{attribute 'GeneratedUsingTerminal: EP8309-0022-0021'}
{attribute addProperty BoxType "EP8309-0022-0021"}
{attribute addProperty Id "Digital_Input_X4_Pin4AT %I*BOOL1Digital_Input_X4_Pin2AT %I*BOOL1Digital_Input_X5_Pin4AT %I*BOOL1Digital_Input_X5_Pin2AT %I*BOOL1Digital_Input_X6_Pin4AT %I*BOOL1Digital_Input_X6_Pin2AT %I*BOOL1Digital_Input_X7_Pin4AT %I*BOOL1Digital_Input_X7_Pin2AT %I*BOOL1"}
{attribute addProperty CRC "1230986660"}
{attribute addProperty Size "8"}
TYPE DIG_Inputs_495F5DA4 EXTENDS InputBase_8311D824 :
STRUCT
	{attribute addProperty Name "Digital_Input_X4_Pin4"}
	Digital_Input_X4_Pin4 AT %I* : BOOL;
	{attribute addProperty Name "Digital_Input_X4_Pin2"}
	Digital_Input_X4_Pin2 AT %I* : BOOL;
	{attribute addProperty Name "Digital_Input_X5_Pin4"}
	Digital_Input_X5_Pin4 AT %I* : BOOL;
	{attribute addProperty Name "Digital_Input_X5_Pin2"}
	Digital_Input_X5_Pin2 AT %I* : BOOL;
	{attribute addProperty Name "Digital_Input_X6_Pin4"}
	Digital_Input_X6_Pin4 AT %I* : BOOL;
	{attribute addProperty Name "Digital_Input_X6_Pin2"}
	Digital_Input_X6_Pin2 AT %I* : BOOL;
	{attribute addProperty Name "Digital_Input_X7_Pin4"}
	Digital_Input_X7_Pin4 AT %I* : BOOL;
	{attribute addProperty Name "Digital_Input_X7_Pin2"}
	Digital_Input_X7_Pin2 AT %I* : BOOL;
END_STRUCT
END_TYPE

(* stored: Version 1.2.0.0, ProductVersion 3.1.4024.9
   DUT DIG_Inputs_495F5DA4: Id {d9581c66-1139-4eb9-a4ce-e5c8797cde0b} *)
